# EPICS StreamDevice protocol: RC3UApp/Db/RC3U.proto
#OutTerminator = CR;
#InTerminator = CR;
Terminator = CR;

watchdog{out ".0101WatchDog%0<sum8>"; in "#01010WatchDog%d%(\$1)d%(\$2)d%(\$3)d%0<sum8>"; wait 1000;}
#ReadContSensor {out ".0102rCtrlSen%0<sum16>"; in "#01020rCtrlSen%d%0<sum8>";}
#ReadsetTemp_read {out ".0103rSetTemp%0<sum8>"; in "#01030rSetTemp%f%0<sum8>";}
#ReadsupTemp_read {out ".0104rSupplyT%0<sum8>"; in "#01040rSupplyT%f%0<sum8>";}
#ReadRetTemp_read {out ".0107rReturnT%0<sum8>"; in "#01070rReturnT%f%0<sum8>";}
#ReadAmbTemp_read {out ".0108rAmbTemp%0<sum8>"; in "#01080rAmbTemp%f%0<sum8>";}
#ReadProcFlow_read {out ".0109rProsFlo%0<sum8>"; in "#01090rProsFlo%f%0<sum8>";}

#SetExtSensorstatus {out ".0112sExtSens%d%0<sum8>"; in "#01120sExtSens%d%0<sum8>";}
#SetChillerStatus {out ".0115sStatus_%d%0<sum8>"; in "#01150sStatus_%d%0<sum8>";}
#Setcontsensor {out ".0116sCtrlSen%d%0<sum8>"; in "#01160sCtrlSen%d%0<sum8>";}
#SetControlTemp_set {out ".0117sCtrlT__%4d%0<sum8>"; in "#01170sCtrlT__%f%0<sum8>";}
